// TIA Portal V20 export
DATA_BLOCK "InstDancerMainDB"   // DB106
// stored: InstanceOfName 2100_DancerMain, InstanceOfType FB
"2100_DancerMain"
   // VAR_INPUT
   //    Enable : Bool;
   //    Stop : Bool;
   //    Reset : Bool;
   //    Parameter : Struct
   //       DancerDirection : Bool;
   //       UnWinderDirection : Bool;
   //       UnwinderTopUse : Bool;
   //       UnwinderBottomUse : Bool;
   //       JogMode : Bool;
   //       SetPoint : LReal;
   //       Input : LReal;
   //       Kp : LReal;
   //       Ki : LReal;
   //       Radius : LReal;
   //    END_STRUCT;
   // END_VAR
   // VAR_OUTPUT
   //    Busy : Struct
   //       TotalBusy : Bool;
   //       EnableBusy : Bool;
   //       StopBusy : Bool;
   //       ResetBusy : Bool;
   //    END_STRUCT;
   //    Done : Struct
   //       TotalDone : Bool;
   //       EnableDone : Bool;
   //       StopDone : Bool;
   //       ResetDone : Bool;
   //    END_STRUCT;
   //    Error : Bool;
   //    ErrorID : DWord;
   //    SubNowStep : DInt;
   //    SubBeforeStep : DInt;
   // END_VAR
   // VAR_IN_OUT
   //    SlaveUnwinderVirtual : DB_ANY;
   //    SlaveUnwinderTop : DB_ANY;
   //    SlaveUnwinderBottom : DB_ANY;
   //    SepaClampX : DB_ANY;
   // END_VAR
   // VAR
   //    statNowCmd : DInt;
   //    statBeforeCmd : DInt;
   //    statDone : Bool;
   //    statTimeTable : Array[1..50] of Time;
   //    statStartTime : Time;
   //    statEndTime : Time;
   //    instTriggerEnable : R_TRIG;
   //    instTriggerStop { S7_SetPoint := 'True'} : R_TRIG;
   //    instTriggerReset { S7_SetPoint := 'True'} : R_TRIG;
   //    instDancerEnable { S7_SetPoint := 'True'} : "2101_DancerEnable";
   //    instDancerStop { S7_SetPoint := 'True'} : "2102_DancerStop";
   //    instDancerReset { S7_SetPoint := 'True'} : "2103_DancerReset";
   // END_VAR
BEGIN
END_DATA_BLOCK
